// TIA Portal project "定时器的学习" (V15.1)

(* hardware
DEVICE "S7-1200 station_1"  S7-1200 Station
   slot 0: "Rack_0"  S7-1200 Rack  Rack  V1.0
   slot 1: "PLC_1"  CPU 1214C DC/DC/DC  6ES7 214-1AG40-0XB0  V4.2
*)

// ===== PLC "PLC_1"  CPU 1214C DC/DC/DC =====

VAR_GLOBAL   // PLC tag table "默认变量表"
   "Tag_1" AT %MD200 : Time;
   "Tag_2" AT %I1.0 : Bool;
   "Tag_3" AT %Q1.0 : Bool;
   "Tag_4" AT %I1.1 : Bool;
   "Tag_5" AT %MD201 : Time;
   "Tag_6" AT %Q1.1 : Bool;
   "Tag_7" AT %I1.3 : Bool;
   "Tag_8" AT %MD202 : Time;
   "Tag_9" AT %Q1.2 : Bool;
   "Tag_10" AT %I1.2 : Bool;
   "Tag_11" AT %I1.4 : Bool;
   "Tag_12" AT %MD203 : Time;
   "Tag_13" AT %Q1.3 : Bool;
END_VAR

// folder: System blocks/Program resources

DATA_BLOCK "IEC_Timer_0_DB"   // DB1
{ S7_Optimized_Access := 'TRUE' }
AUTHOR : Simatic
FAMILY : IEC
NAME : IEC_TMR
VERSION : 1.0
// stored: InstanceOfName IEC_TIMER
"IEC_TIMER"
BEGIN
END_DATA_BLOCK

DATA_BLOCK "IEC_Timer_0_DB_1"   // DB2
{ S7_Optimized_Access := 'TRUE' }
AUTHOR : Simatic
FAMILY : IEC
NAME : IEC_TMR
VERSION : 1.0
// stored: InstanceOfName IEC_TIMER
"IEC_TIMER"
BEGIN
END_DATA_BLOCK

DATA_BLOCK "IEC_Timer_0_DB_2"   // DB3
{ S7_Optimized_Access := 'TRUE' }
AUTHOR : Simatic
FAMILY : IEC
NAME : IEC_TMR
VERSION : 1.0
// stored: InstanceOfName IEC_TIMER
"IEC_TIMER"
BEGIN
END_DATA_BLOCK

DATA_BLOCK "IEC_Timer_0_DB_3"   // DB4
{ S7_Optimized_Access := 'TRUE' }
AUTHOR : Simatic
FAMILY : IEC
NAME : IEC_TMR
VERSION : 1.0
// stored: InstanceOfName IEC_TIMER
"IEC_TIMER"
BEGIN
END_DATA_BLOCK

// folder: (top level)

ORGANIZATION_BLOCK "Main"   // OB1, LAD, ProgramCycle
TITLE = "Main Program Sweep (Cycle)"
{ S7_Optimized_Access := 'TRUE' }
VERSION : 0.1
   VAR_INPUT
      Initial_Call : Bool;   // Initial call of this OB
      Remanence : Bool;   // =True, if remanent data are available
   END_VAR
BEGIN

REGION Network 1
   // 脉冲定时器
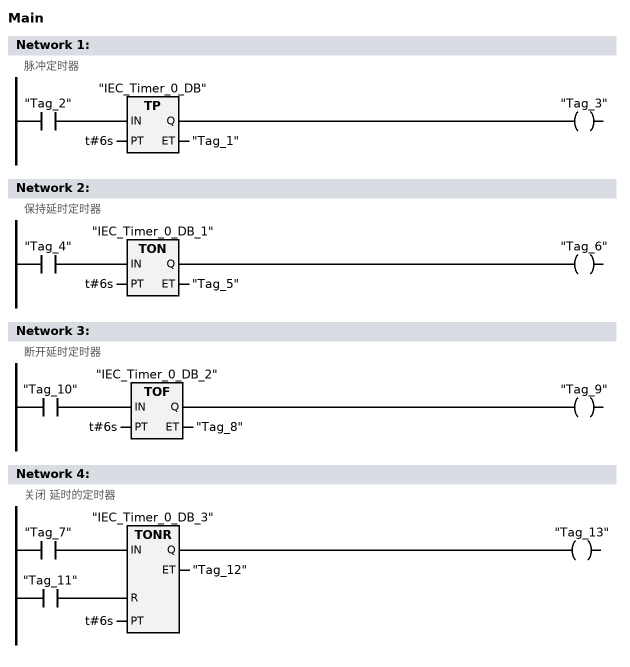
   "IEC_Timer_0_DB".TP(IN := "Tag_2", PT := t#6s, ET => "Tag_1");
   "Tag_3" := "IEC_Timer_0_DB".Q;
END_REGION

REGION Network 2
   // 保持延时定时器
   "IEC_Timer_0_DB_1".TON(IN := "Tag_4", PT := t#6s, ET => "Tag_5");
   "Tag_6" := "IEC_Timer_0_DB_1".Q;
END_REGION

REGION Network 3
   // 断开延时定时器
   "IEC_Timer_0_DB_2".TOF(IN := "Tag_10", PT := t#6s, ET => "Tag_8");
   "Tag_9" := "IEC_Timer_0_DB_2".Q;
END_REGION

REGION Network 4
   // 关闭 延时的定时器
   "IEC_Timer_0_DB_3".TONR(IN := "Tag_7", R := "Tag_11", PT := t#6s, ET => "Tag_12");
   "Tag_13" := "IEC_Timer_0_DB_3".Q;
END_REGION
END_ORGANIZATION_BLOCK